FUNCTION_BLOCK TemplateSimple (* Example for a Simple Function Block Type *)
  (* Standard: 61499-1 *)
  (* Version 0.0, 2018-10-15, Peter Gsellmann, TU Wien/ACIN *)
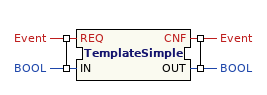
  EVENT_INPUT
    REQ WITH IN; (* Normal Execution Request *)
  END_EVENT
  EVENT_OUTPUT
    CNF WITH OUT; (* Execution Confirmation *)
  END_EVENT
  VAR_INPUT
    IN : BOOL; (* Input *)
  END_VAR
  VAR_OUTPUT
    OUT : BOOL; (* Output *)
  END_VAR
  EC_STATES
    REQ : REQ -> CNF;
  END_STATES
  ALGORITHM REQ IN ST: (* Executed algorithm *)
OUT := IN;
  END_ALGORITHM
END_FUNCTION_BLOCK
